(* CoDeSys 2.3.9.47 project: gym_2016_12_27_1.pr6 *)
(* Libraries: PlcSystemBC.lb6 21.3.01 10:03:02, PlcHelperBC.lb6 7.5.01 10:03:00, TcAdsBC.lb6 5.7.02 10:03:02, standard.lib 5.6.98 10:03:02, TcBABasic.lib 22.7.15 14:46:14, TcPlcUtilitiesBC.lb6 13.5.05 10:19:40 *)

(* Global variable list: main *)
VAR_GLOBAL
	dataDerevo: ARRAY[0..3] OF BYTE;
	dataDerevo_prev :ARRAY[0..3] OF BYTE;

	ads_adr_derevo: STRING:='10.0.5.64.1.1';

	write_ads: ADSWRITE;

	bDarkOutside						AT%MX0.0:BOOL;


	iHour							AT%MB1:	BYTE;
	iMinute							AT%MB3:	BYTE;

	t_out							AT%MB6 :	 REAL;

	eib_gym01 						AT %MX10.0:	 BOOL;
	eib_gym02 						AT %MX10.1:	 BOOL;
	eib_training01 					AT %MX10.2:	 BOOL;
	eib_training02						AT %MX10.3:	 BOOL;
	eib_training03						AT %MX10.4:	 BOOL;
	eib_gym_stairs_bra				AT %MX10.5:	 BOOL;
	eib_pool_hall_spotlight				AT %MX10.6:	 BOOL;
	eib_pool_hall_LED				AT %MX10.7:	 BOOL;

	eib_pool_light 					AT %MX11.0:	 BOOL;
	eib_sphere_ceiling_light 			AT %MX11.1:	 BOOL;
	eib_sphere_light 					AT %MX11.2:	 BOOL;
	eib_gym_cinema_bra 				AT %MX11.3:	 BOOL;
	eib_gym_shower01_light			AT %MX11.4:	 BOOL;
	eib_gym_shower02_light			AT %MX11.5:	 BOOL;
	eib_gym_corridor_light				AT %MX11.6:	 BOOL;
	eib_gym_stairs_light 				AT %MX11.7:	 BOOL;

	eib_gym_WC_light 				AT %MX12.0:	 BOOL;
	eib_cinema_temporary_light		AT %MX12.1:	 BOOL;





END_VAR

(* Global variable list: physical *)
(* @GLOBAL_VARIABLE_LIST := TwinCAT_Import *)
(* @PATH := '' *)
VAR_GLOBAL (* DO NOT CHANGE THIS SHEET MANUALLY! *)
	PlcInVar_0	AT %QB128:	USINT;
	PlcInVar_1	AT %QB129:	USINT;
	PlcInVar_2	AT %QB130:	USINT;
	PlcInVar_3	AT %QB131:	USINT;
	PlcInVar_4	AT %QB132:	USINT;
	PlcInVar_5	AT %QB133:	USINT;
	PlcInVar_6	AT %QB134:	USINT;
	PlcInVar_7	AT %QB135:	USINT;
	PlcInVar_8	AT %QB136:	USINT;
	PlcInVar_9	AT %QB137:	USINT;
	PlcInVar_10	AT %QB138:	USINT;
	PlcInVar_11	AT %QB139:	USINT;
	PlcInVar_12	AT %QB140:	USINT;
	PlcInVar_13	AT %QB141:	USINT;
	PlcInVar_14	AT %QB142:	USINT;
	PlcInVar_15	AT %QB143:	USINT;
	PlcOutVar_0	AT %IB128:	USINT;
	PlcOutVar_1	AT %IB129:	USINT;
	PlcOutVar_2	AT %IB130:	USINT;
	PlcOutVar_3	AT %IB131:	USINT;
	PlcOutVar_4	AT %IB132:	USINT;
	PlcOutVar_5	AT %IB133:	USINT;
	PlcOutVar_6	AT %IB134:	USINT;
	PlcOutVar_7	AT %IB135:	USINT;
	PlcOutVar_8	AT %IB136:	USINT;
	PlcOutVar_9	AT %IB137:	USINT;
	PlcOutVar_10	AT %IB138:	USINT;
	PlcOutVar_11	AT %IB139:	USINT;
	PlcOutVar_12	AT %IB140:	USINT;
	PlcOutVar_13	AT %IB141:	USINT;
	PlcOutVar_14	AT %IB142:	USINT;
	PlcOutVar_15	AT %IB143:	USINT;
	gym01_light				AT %QX0.0:	BOOL; (*K01*)
	training03_light			AT %QX0.1:	BOOL; (*K05*)
	gym02_light				AT %QX0.2:	BOOL; (*K02*)
	gym_stairs_bra_right		AT %QX0.3:	BOOL; (*K06*)
	training01_light			AT %QX0.4:	BOOL; (*K03*)
	gym_stairs_bra_left		AT %QX0.5:	BOOL; (*K07*)
	training02_light			AT %QX0.6:	BOOL; (*K04*)
	pool_hall_spotlight		AT %QX0.7:	BOOL; (*K08*)

	pool_hall_ceiling_LED	AT %QX1.0:	BOOL; (*K09*)
	pool_light				AT %QX1.1:	BOOL; (*K13*)
	sphere_ceiling_light		AT %QX1.2:	BOOL; (*K10*)
	gym03_light				AT %QX1.3:	BOOL; (*K14*)
	sphere_light01			AT %QX1.4:	BOOL; (*K11*)
	gym04_light				AT %QX1.5:	BOOL; (*K15*)
	gym_cinema_bra		AT %QX1.6:	BOOL; (*K12*)
	training04_light			AT %QX1.7:	BOOL; (*K16*)

	training05_light			AT %QX2.0:	BOOL; (*K17*)
	gym_shower01_light		AT %QX2.1:	BOOL; (*K21*)
	training06_light			AT %QX2.2:	BOOL; (*K18*)
	gym_shower02_light		AT %QX2.3:	BOOL; (*K22*)
	gym_WC_corridor		AT %QX2.4:	BOOL; (*K19*)
	gym_stairs_light			AT %QX2.5:	BOOL; (*K23*)
	gym_WC_light			AT %QX2.6:	BOOL; (*K20*)
	sphere_light02			AT %QX2.7:	BOOL; (*K24*)

	pool_hall_LED			AT %QX3.0:	BOOL; (*K25*)
	Term_5_KL2408_2_Output	AT %QX3.1:	BOOL;
	gym_cinema_TEMPORARY_light	AT %QX3.2:	BOOL; (*K26*)


	Term_5_KL2408_4_Output	AT %QX3.3:	BOOL;
	Term_5_KL2408_5_Output	AT %QX3.4:	BOOL;
	Term_5_KL2408_6_Output	AT %QX3.5:	BOOL;
	Term_5_KL2408_7_Output	AT %QX3.6:	BOOL;
	Term_5_KL2408_8_Output	AT %QX3.7:	BOOL;

	Term_6_KL1408_1_Input	AT %IX0.0:	BOOL;
	sw_01_1_2	AT %IX0.1:	BOOL;
	Term_6_KL1408_3_Input	AT %IX0.2:	BOOL;
	Term_6_KL1408_4_Input	AT %IX0.3:	BOOL;
	Term_6_KL1408_5_Input	AT %IX0.4:	BOOL;
	sw_01_1_1	AT %IX0.5:	BOOL;
	sw_01_2_1	AT %IX0.6:	BOOL;

	sw_07_1_1			AT %IX0.7:	BOOL;

	sw_07_2_1			AT %IX1.0:	BOOL;
	sw_14_1_1			AT %IX1.1:	BOOL;
	Term_7_KL1408_3_Input	AT %IX1.2:	BOOL;
	sw_14_1_2			AT %IX1.3:	BOOL;
	Term_7_KL1408_5_Input	AT %IX1.4:	BOOL;
	sw_14_2_2			AT %IX1.5:	BOOL;
	Term_7_KL1408_7_Input	AT %IX1.6:	BOOL;
	sw_14_2_1			AT %IX1.7:	BOOL;

	sw_14_3_1			AT %IX2.0:	BOOL;
	sw_09_2_2			AT %IX2.1:	BOOL;
	sw_14_3_2			AT %IX2.2:	BOOL;
	sw_09_3_1			AT %IX2.3:	BOOL;
	sw_09_1_1			AT %IX2.4:	BOOL;
	sw_09_3_2			AT %IX2.5:	BOOL;
	sw_09_2_1			AT %IX2.6:	BOOL;
	sw_09_1_2			AT %IX2.7:	BOOL;

	sw_04_1				AT %IX3.0:	BOOL;
	Term_9_KL1408_2_Input	AT %IX3.1:	BOOL;
	sw_04_2				AT %IX3.2:	BOOL;
	Term_9_KL1408_4_Input	AT %IX3.3:	BOOL;
	sw_06_1				AT %IX3.4:	BOOL;
	Term_9_KL1408_6_Input	AT %IX3.5:	BOOL;
	sw_06_2				AT %IX3.6:	BOOL;
	Term_9_KL1408_8_Input	AT %IX3.7:	BOOL;
	Term_10_KL1408_1_Input	AT %IX4.0:	BOOL;
	Term_10_KL1408_2_Input	AT %IX4.1:	BOOL;
	Term_10_KL1408_3_Input	AT %IX4.2:	BOOL;
	Term_10_KL1408_4_Input	AT %IX4.3:	BOOL;
	Term_10_KL1408_5_Input	AT %IX4.4:	BOOL;
	Term_10_KL1408_6_Input	AT %IX4.5:	BOOL;
	Term_10_KL1408_7_Input	AT %IX4.6:	BOOL;
	Term_10_KL1408_8_Input	AT %IX4.7:	BOOL;
END_VAR

(* @OBJECT_END := TwinCAT_Import *)

(* POU MAIN, ST *)
PROGRAM MAIN
VAR
	i,j:INT;
	write:BOOL;
	heartBeat: TP;
END_VAR
heartBeat(IN:= NOT heartBeat.Q, PT:=t#5s);
Light;
(*Counters;*)
write_dataDerevo;
ADS_Communication;
END_PROGRAM
ACTION write_dataDerevo:
	dataDerevo[0].0:= gym01_light ;
	dataDerevo[0].1:= gym02_light;
	dataDerevo[0].2:= training01_light;
	dataDerevo[0].3:= training02_light;
	dataDerevo[0].4:= training03_light;
	dataDerevo[0].5:= gym_stairs_bra_left;
	dataDerevo[0].6:= pool_hall_spotlight;
	dataDerevo[0].7:= pool_hall_LED;

	dataDerevo[1].0:= pool_light;
	dataDerevo[1].1:= sphere_ceiling_light;
	dataDerevo[1].2:= sphere_light01;
	dataDerevo[1].3:= gym_cinema_bra;
	dataDerevo[1].4:= gym_shower01_light;
	dataDerevo[1].5:= gym_shower02_light;
	dataDerevo[1].6:= gym_WC_corridor;
	dataDerevo[1].7:= gym_stairs_light;

	dataDerevo[2].0:= gym_WC_light;



FOR i:=0 TO (SIZEOF(dataDerevo))-1 DO
	IF dataDerevo[i]<>dataDerevo_prev[i]  THEN
		write:=TRUE;
		EXIT;
	ELSE
		write:=FALSE;
	END_IF
END_FOR


FOR j:=0 TO (SIZEOF(dataDerevo))-1 DO
	dataDerevo_prev[j]:=dataDerevo[j];
END_FOR
END_ACTION

(* POU Light, CFC *)
PROGRAM Light
VAR
	fb_gym01_light			: FB_Light;
	fb_gym02_light			: FB_Light;
	fb_training01_light		: FB_Light;
	fb_training02_light		: FB_Light;
	fb_training03_light		: FB_Light;
	fb_gym_stairs_bra		: FB_Light;
	fb_pool_hall_spotlight	: FB_Light;
	fb_pool_hall_LED		: FB_Light;
	fb_pool_light			: FB_Light;
	fb_sphere_ceiling_light	: FB_Light;
	fb_sphere_light			: FB_Light;
	fb_gym_cinema_bra		: FB_Light;
	fb_gym_shower01_light	: FB_Light;
	fb_gym_shower02_light	: FB_Light;
	fb_gym_corridor_light	: FB_Light;
	fb_gym_stairs_light		: FB_Light;
	fb_gym_WC_light		: FB_Light;


	fb_cinema_temporary_light	:FB_Light;

END_VAR
VAR (* helpers for the ST form of the networks *)
	_t99 : BOOL;
	_t101 : BOOL;
	_t104 : BOOL;
END_VAR
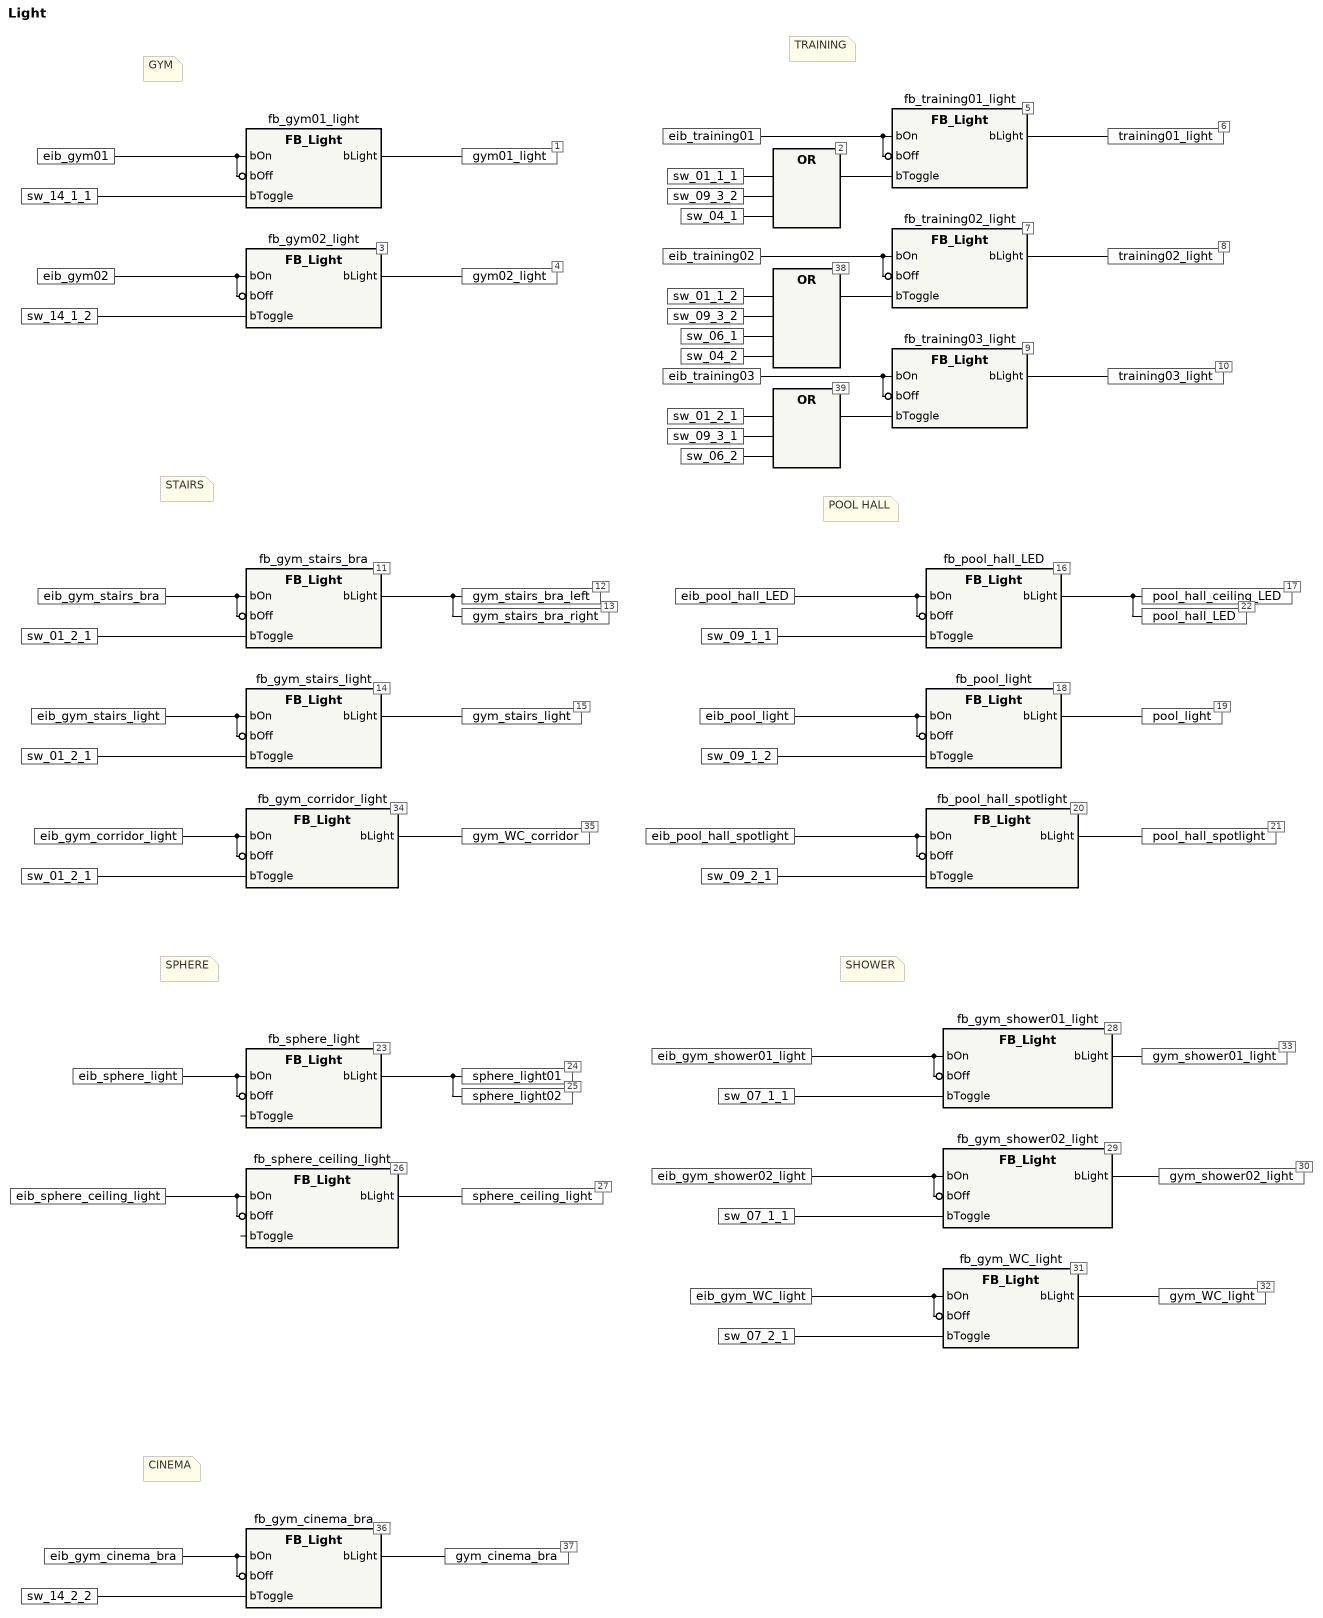
_CFC_ (* Continuous Function Chart, elements in execution order *)
(* GYM *)
#0 fb_gym01_light:FB_Light(bOn: eib_gym01, bOff: NOT eib_gym01, bToggle: sw_14_1_1)
#1 gym01_light <= #0.bLight
#2 OR(sw_01_1_1, sw_09_3_2, sw_04_1)
#3 fb_gym02_light:FB_Light(bOn: eib_gym02, bOff: NOT eib_gym02, bToggle: sw_14_1_2)
#4 gym02_light <= #3.bLight
(* TRAINING *)
(* STAIRS *)
#5 fb_training01_light:FB_Light(bOn: eib_training01, bOff: NOT eib_training01, bToggle: #2)
#6 training01_light <= #5.bLight
#7 fb_training02_light:FB_Light(bOn: eib_training02, bOff: NOT eib_training02, bToggle: #38)
#8 training02_light <= #7.bLight
#9 fb_training03_light:FB_Light(bOn: eib_training03, bOff: NOT eib_training03, bToggle: #39)
#10 training03_light <= #9.bLight
#11 fb_gym_stairs_bra:FB_Light(bOn: eib_gym_stairs_bra, bOff: NOT eib_gym_stairs_bra, bToggle: sw_01_2_1)
#12 gym_stairs_bra_left <= #11.bLight
#13 gym_stairs_bra_right <= #11.bLight
#14 fb_gym_stairs_light:FB_Light(bOn: eib_gym_stairs_light, bOff: NOT eib_gym_stairs_light, bToggle: sw_01_2_1)
#15 gym_stairs_light <= #14.bLight
(* POOL HALL *)
#16 fb_pool_hall_LED:FB_Light(bOn: eib_pool_hall_LED, bOff: NOT eib_pool_hall_LED, bToggle: sw_09_1_1)
#17 pool_hall_ceiling_LED <= #16.bLight
#18 fb_pool_light:FB_Light(bOn: eib_pool_light, bOff: NOT eib_pool_light, bToggle: sw_09_1_2)
#19 pool_light <= #18.bLight
#20 fb_pool_hall_spotlight:FB_Light(bOn: eib_pool_hall_spotlight, bOff: NOT eib_pool_hall_spotlight, bToggle: sw_09_2_1)
#21 pool_hall_spotlight <= #20.bLight
#22 pool_hall_LED <= #16.bLight
(* SPHERE *)
#23 fb_sphere_light:FB_Light(bOn: eib_sphere_light, bOff: NOT eib_sphere_light, bToggle: -)
#24 sphere_light01 <= #23.bLight
#25 sphere_light02 <= #23.bLight
#26 fb_sphere_ceiling_light:FB_Light(bOn: eib_sphere_ceiling_light, bOff: NOT eib_sphere_ceiling_light, bToggle: -)
#27 sphere_ceiling_light <= #26.bLight
(* SHOWER *)
#28 fb_gym_shower01_light:FB_Light(bOn: eib_gym_shower01_light, bOff: NOT eib_gym_shower01_light, bToggle: sw_07_1_1)
#29 fb_gym_shower02_light:FB_Light(bOn: eib_gym_shower02_light, bOff: NOT eib_gym_shower02_light, bToggle: sw_07_1_1)
#30 gym_shower02_light <= #29.bLight
#31 fb_gym_WC_light:FB_Light(bOn: eib_gym_WC_light, bOff: NOT eib_gym_WC_light, bToggle: sw_07_2_1)
#32 gym_WC_light <= #31.bLight
#33 gym_shower01_light <= #28.bLight
#34 fb_gym_corridor_light:FB_Light(bOn: eib_gym_corridor_light, bOff: NOT eib_gym_corridor_light, bToggle: sw_01_2_1)
#35 gym_WC_corridor <= #34.bLight
(* CINEMA *)
#36 fb_gym_cinema_bra:FB_Light(bOn: eib_gym_cinema_bra, bOff: NOT eib_gym_cinema_bra, bToggle: sw_14_2_2)
#37 gym_cinema_bra <= #36.bLight
#38 OR(sw_01_1_2, sw_09_3_2, sw_06_1, sw_04_2)
#39 OR(sw_01_2_1, sw_09_3_1, sw_06_2)
_END_CFC_
(* the same logic as Structured Text *)
(* GYM *)
fb_gym01_light(bOn := eib_gym01, bOff := NOT eib_gym01, bToggle := sw_14_1_1);
gym01_light := fb_gym01_light.bLight;
_t99 := sw_01_1_1 OR sw_09_3_2 OR sw_04_1;
fb_gym02_light(bOn := eib_gym02, bOff := NOT eib_gym02, bToggle := sw_14_1_2);
gym02_light := fb_gym02_light.bLight;
(* TRAINING *)
(* STAIRS *)
fb_training01_light(bOn := eib_training01, bOff := NOT eib_training01, bToggle := _t99);
training01_light := fb_training01_light.bLight;
fb_training02_light(bOn := eib_training02, bOff := NOT eib_training02, bToggle := _t101);
training02_light := fb_training02_light.bLight;
fb_training03_light(bOn := eib_training03, bOff := NOT eib_training03, bToggle := _t104);
training03_light := fb_training03_light.bLight;
fb_gym_stairs_bra(bOn := eib_gym_stairs_bra, bOff := NOT eib_gym_stairs_bra, bToggle := sw_01_2_1);
gym_stairs_bra_left := fb_gym_stairs_bra.bLight;
gym_stairs_bra_right := fb_gym_stairs_bra.bLight;
fb_gym_stairs_light(bOn := eib_gym_stairs_light, bOff := NOT eib_gym_stairs_light, bToggle := sw_01_2_1);
gym_stairs_light := fb_gym_stairs_light.bLight;
(* POOL HALL *)
fb_pool_hall_LED(bOn := eib_pool_hall_LED, bOff := NOT eib_pool_hall_LED, bToggle := sw_09_1_1);
pool_hall_ceiling_LED := fb_pool_hall_LED.bLight;
fb_pool_light(bOn := eib_pool_light, bOff := NOT eib_pool_light, bToggle := sw_09_1_2);
pool_light := fb_pool_light.bLight;
fb_pool_hall_spotlight(bOn := eib_pool_hall_spotlight, bOff := NOT eib_pool_hall_spotlight, bToggle := sw_09_2_1);
pool_hall_spotlight := fb_pool_hall_spotlight.bLight;
pool_hall_LED := fb_pool_hall_LED.bLight;
(* SPHERE *)
fb_sphere_light(bOn := eib_sphere_light, bOff := NOT eib_sphere_light);
sphere_light01 := fb_sphere_light.bLight;
sphere_light02 := fb_sphere_light.bLight;
fb_sphere_ceiling_light(bOn := eib_sphere_ceiling_light, bOff := NOT eib_sphere_ceiling_light);
sphere_ceiling_light := fb_sphere_ceiling_light.bLight;
(* SHOWER *)
fb_gym_shower01_light(bOn := eib_gym_shower01_light, bOff := NOT eib_gym_shower01_light, bToggle := sw_07_1_1);
fb_gym_shower02_light(bOn := eib_gym_shower02_light, bOff := NOT eib_gym_shower02_light, bToggle := sw_07_1_1);
gym_shower02_light := fb_gym_shower02_light.bLight;
fb_gym_WC_light(bOn := eib_gym_WC_light, bOff := NOT eib_gym_WC_light, bToggle := sw_07_2_1);
gym_WC_light := fb_gym_WC_light.bLight;
gym_shower01_light := fb_gym_shower01_light.bLight;
fb_gym_corridor_light(bOn := eib_gym_corridor_light, bOff := NOT eib_gym_corridor_light, bToggle := sw_01_2_1);
gym_WC_corridor := fb_gym_corridor_light.bLight;
(* CINEMA *)
fb_gym_cinema_bra(bOn := eib_gym_cinema_bra, bOff := NOT eib_gym_cinema_bra, bToggle := sw_14_2_2);
gym_cinema_bra := fb_gym_cinema_bra.bLight;
_t101 := sw_01_1_2 OR sw_09_3_2 OR sw_06_1 OR sw_04_2;
_t104 := sw_01_2_1 OR sw_09_3_1 OR sw_06_2;
END_PROGRAM

(* POU ADS_Communication, CFC *)
PROGRAM ADS_Communication
VAR
	fb_DerevoADSwrite: ADSWRITE;


	counter_error,counter_busy: CTU;
END_VAR
VAR (* helpers for the ST form of the networks *)
	_t21 : DWORD;
	_t23 : DWORD;
	_t42 : BOOL;
END_VAR
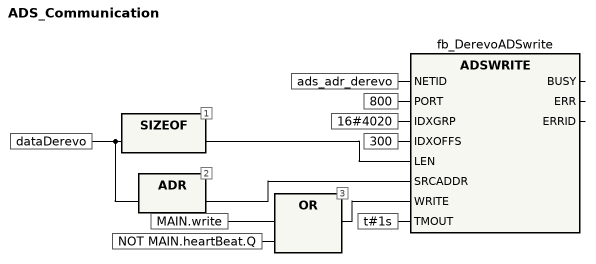
_CFC_ (* Continuous Function Chart, elements in execution order *)
#0 fb_DerevoADSwrite:ADSWRITE(NETID: ads_adr_derevo, PORT: 800, IDXGRP: 16#4020, IDXOFFS: 300, LEN: #1, SRCADDR: #2, WRITE: #3, TMOUT: t#1s)
#1 SIZEOF(dataDerevo)
#2 ADR(dataDerevo)
#3 OR(MAIN.write, NOT MAIN.heartBeat.Q)
_END_CFC_
(* the same logic as Structured Text *)
fb_DerevoADSwrite(NETID := ads_adr_derevo, PORT := 800, IDXGRP := 16#4020, IDXOFFS := 300, LEN := _t21, SRCADDR := _t23, WRITE := _t42, TMOUT := t#1s);
_t21 := SIZEOF(dataDerevo);
_t23 := ADR(dataDerevo);
_t42 := MAIN.write OR NOT MAIN.heartBeat.Q;
END_PROGRAM

(* POU Counters, ST *)
PROGRAM Counters
VAR

	counter_6_KL1408_1_Input : CTU;

	counter_6_KL1408_3_Input	:	CTU;
	counter_6_KL1408_4_Input	:	CTU;
	counter_6_KL1408_5_Input	:	CTU;
	counter_6_KL1408_6_Input	:	CTU;

	counter_6_KL1408_8_Input	:	CTU;
	counter_7_KL1408_1_Input	:	CTU;
	counter_7_KL1408_2_Input	:	CTU;
	counter_7_KL1408_3_Input	:	CTU;
	counter_7_KL1408_4_Input	:	CTU;
	counter_7_KL1408_5_Input	:	CTU;
	counter_7_KL1408_6_Input	:	CTU;
	counter_7_KL1408_7_Input	:	CTU;
	counter_7_KL1408_8_Input	:	CTU;
	counter_8_KL1408_1_Input	:	CTU;
	counter_8_KL1408_2_Input	:	CTU;
	counter_8_KL1408_3_Input	:	CTU;
	counter_8_KL1408_4_Input	:	CTU;
	counter_8_KL1408_5_Input	:	CTU;
	counter_8_KL1408_6_Input	:	CTU;
	counter_8_KL1408_7_Input	:	CTU;
	counter_8_KL1408_8_Input	:	CTU;
	counter_9_KL1408_1_Input	:	CTU;
	counter_9_KL1408_2_Input	:	CTU;
	counter_9_KL1408_3_Input	:	CTU;
	counter_9_KL1408_4_Input	:	CTU;
	counter_9_KL1408_5_Input	:	CTU;
	counter_9_KL1408_6_Input	:	CTU;
	counter_9_KL1408_7_Input	:	CTU;
	counter_9_KL1408_8_Input	:	CTU;
	counter_10_KL1408_1_Input	:	CTU;
	counter_10_KL1408_2_Input	:	CTU;
	counter_10_KL1408_3_Input	:	CTU;
	counter_10_KL1408_4_Input	:	CTU;
	counter_10_KL1408_5_Input	:	CTU;
	counter_10_KL1408_6_Input	:	CTU;
	counter_10_KL1408_7_Input	:	CTU;
	counter_10_KL1408_8_Input	:	CTU;

	sw01 : INT;
	sw02 : INT;
	sw03 : INT;
	sw04 : INT;
	sw05 : INT;
	sw06 : INT;
	sw07 : INT;
	sw08 : INT;
	sw09 : INT;
	sw10 : INT;
	sw11 : INT;
	sw12 : INT;
	sw13 : INT;
	sw14 : INT;
	sw15 : INT;
	sw16 : INT;
	sw17 : INT;
	sw18 : INT;
	sw19 : INT;
	sw20 : INT;
	sw21 : INT;
	sw22 : INT;
	sw23 : INT;
	sw24 : INT;
	sw25 : INT;
	sw26 : INT;
	sw27 : INT;
	sw28 : INT;
	sw29 : INT;
	sw30 : INT;
	sw31 : INT;
	sw32 : INT;
	sw33 : INT;
	sw34 : INT;
	sw35 : INT;
	sw36 : INT;
	sw37 : INT;
	sw38 : INT;
	sw39 : INT;


END_VAR
	counter_6_KL1408_1_Input(CU:= Term_6_KL1408_1_Input, CV=>sw01);

	counter_6_KL1408_3_Input(CU:= Term_6_KL1408_3_Input, CV=>sw02);
	counter_6_KL1408_4_Input(CU:= Term_6_KL1408_4_Input, CV=>sw03);
	counter_6_KL1408_5_Input(CU:= Term_6_KL1408_5_Input, CV=>sw04);





	counter_7_KL1408_3_Input(CU:= Term_7_KL1408_3_Input, CV=>sw09);

	counter_7_KL1408_5_Input(CU:= Term_7_KL1408_5_Input, CV=>sw11);

	counter_7_KL1408_7_Input(CU:= Term_7_KL1408_7_Input, CV=>sw13);












	counter_9_KL1408_2_Input(CU:= Term_9_KL1408_2_Input, CV=>sw24);

	counter_9_KL1408_4_Input(CU:= Term_9_KL1408_4_Input, CV=>sw26);

	counter_9_KL1408_6_Input(CU:= Term_9_KL1408_6_Input, CV=>sw28);

	counter_9_KL1408_8_Input(CU:= Term_9_KL1408_8_Input, CV=>sw30);

	counter_10_KL1408_1_Input(CU:= Term_10_KL1408_1_Input, CV=>sw31);
	counter_10_KL1408_2_Input(CU:= Term_10_KL1408_2_Input, CV=>sw32);
	counter_10_KL1408_3_Input(CU:= Term_10_KL1408_3_Input, CV=>sw33);
	counter_10_KL1408_4_Input(CU:= Term_10_KL1408_4_Input, CV=>sw34);
	counter_10_KL1408_5_Input(CU:= Term_10_KL1408_5_Input, CV=>sw35);
	counter_10_KL1408_6_Input(CU:= Term_10_KL1408_6_Input, CV=>sw36);
	counter_10_KL1408_7_Input(CU:= Term_10_KL1408_7_Input, CV=>sw37);
	counter_10_KL1408_8_Input(CU:= Term_10_KL1408_8_Input, CV=>sw38);
END_PROGRAM
